TYPE ST_SafetyGroup :
STRUCT
END_STRUCT
END_TYPE

(* stored: Version 1.1.0.1, ProductVersion 3.1.4024.11
   DUT ST_SafetyGroup: Id {a9f34797-5888-4753-bba8-661e2dab047a} *)
